// TIA Portal V20 export
FUNCTION_BLOCK "CC_Hydraulic_Rollers"   // FB101, LAD
{ S7_Optimized_Access := 'TRUE' }
// stored: AutoNumber false, MemoryReserve 100, SetENOAutomatically false
   VAR_INPUT
      ReqUp : Bool;
      ReqDown : Bool;
      Sensor1Down : Bool;
      Sensor1Up : Bool;
      Sensor2Down : Bool;
      Sensor2Up : Bool;
      InterlockMove : Bool;
      HydUnitReady : Bool;
   END_VAR
   VAR_OUTPUT
      HydraulicUnit : Bool;
      ValveUp : Bool;
      ValveDown : Bool;
      error : Byte;   // %X0 – nieprawidłowa pozycja dolna %X1 nieprawidłowa pozycja górna %X2 – przekroczony czas ruchu
      "Step" : Int;
      PosUp : Bool;
      PosDown : Bool;
   END_VAR
   VAR
      IEC_Extention { S7_SetPoint := 'True'} : TON_TIME;
      IEC_RETRACTION { S7_SetPoint := 'True'} : TON_TIME;
      tMotionTimeout { S7_SetPoint := 'True'} : TON_TIME;
   END_VAR
   VAR CONSTANT
      STEP_RETRACT : Int := 1;
      STEP_MOVING : Int := 2;
      STEP_EXTEND : Int := 3;
   END_VAR
BEGIN

REGION Network 1: ValveUp
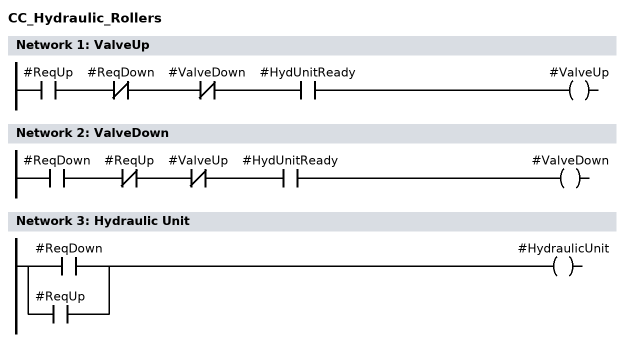
   RUNG wire#powerrail
      Contact( #ReqUp )
      I_Contact( #ReqDown )
      I_Contact( #ValveDown )
      Contact( #HydUnitReady )
      Coil( #ValveUp )
   END_RUNG
   // the same network as SCL:
   #ValveUp := #ReqUp AND NOT #ReqDown AND NOT #ValveDown AND #HydUnitReady;
END_REGION

REGION Network 2: ValveDown
   RUNG wire#powerrail
      Contact( #ReqDown )
      I_Contact( #ReqUp )
      I_Contact( #ValveUp )
      Contact( #HydUnitReady )
      Coil( #ValveDown )
   END_RUNG
   // the same network as SCL:
   #ValveDown := #ReqDown AND NOT #ReqUp AND NOT #ValveUp AND #HydUnitReady;
END_REGION

REGION Network 3: Hydraulic Unit
   RUNG wire#powerrail
      Contact( #ReqDown )
      wire#w1
      Coil( #HydraulicUnit )
   END_RUNG
   RUNG wire#powerrail
      Contact( #ReqUp )
   END_RUNG wire#w1
   // the same network as SCL:
   #HydraulicUnit := #ReqDown OR #ReqUp;
END_REGION

REGION Network 4 (SCL)
   #PosDown := false;
   #PosUp := FALSE;
   #Step := 0;
   IF #Sensor1Down = 0 AND #Sensor1Up = 1 AND #Sensor2Down = 0 AND #Sensor2Up = 1 THEN
       #Step.%X3 := TRUE;
       #PosUp := True;
   ELSIF #Sensor1Down = 1 AND #Sensor1Up =0 AND #Sensor2Down =1 AND #Sensor2Up =0 THEN
       #Step.%X1:= TRUE;
       #PosDown := True;
   ELSE
       #Step.%X2 := TRUE;
   END_IF;
END_REGION
END_FUNCTION_BLOCK
